TYPE ST_HMIEButton_HMI_Link EXTENDS ST_BaseComponent_HMI_Link :
STRUCT
	stButtonHMI			: ST_HMIEButton_HMI;
END_STRUCT
END_TYPE

(* stored: Version 1.1.0.1
   DUT ST_HMIEButton_HMI_Link: Id {8c4ec469-8bd9-016d-035f-17b632626697} *)
